// TIA Portal V19 export
TYPE "ValveConfig"
// stored: Access Published
   STRUCT
      RestLimSwitchExist : Bool;   // Rest limit switch exist
      WorkLimSwitchExist : Bool;   // Work limit switch exist
      CheckOilInPressure : Bool;   // Use for oil valve
      CutRestWhenIsAtRest : Bool;   // Cut rest command when valve is at rest
      CutWorkWhenIsAtWork : Bool;   // Cut work command when valve is at work
      RestTime : Time;   // Time or delay for rest position (depend if limit switch esxist)
      WorkTime : Time;   // Time or delay for work position (depend if limit switch esxist)
      RestTimeOut : Time;   // Time out of rest command
      WorkTimeOut : Time;   // Time out of work command
   END_STRUCT;
END_TYPE
